SUBAPPLICATION StartStopDemo (* Start/Stop pattern demo: E_SR (persistent start/stop state) gates E_PERMIT, which in turn gates TrueUntil.TRIGGER *)
  (* Standard: 61499-2; Description: Copyright (c) 2026 Meisterschulen am Ostbahnhof This program and the accompanying materials are made available under the terms of the Eclipse Public License 2.0 which is available at https://www.eclipse.org/legal/epl-2.0/ SPDX-License-Identifier: EPL-2.0 *)
  (* Version 1.0, 2026-08-31, Franz Höpfinger, Meisterschulen am Ostbahnhof, Start/Stop design pattern (IEC 61499 primer course, Module 6, Valeriy Vyatkin, slide 70), demo application *)
  PACKAGE Meins::DesingPatterns::StartStopPattern;
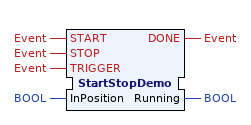
  EVENT_INPUT
    START; (* Start the plant: opens the permit gate *)
    STOP; (* Stop the plant: closes the permit gate *)
    TRIGGER; (* Ask the step to run - only actually reaches it while the plant is started *)
  END_EVENT
  EVENT_OUTPUT
    DONE; (* The step completed (only fires if the plant was started when TRIGGER arrived) *)
  END_EVENT
  VAR_INPUT
    InPosition : BOOL; (* Demo: simulate the step's actuator reaching its position *)
  END_VAR
  VAR_OUTPUT
    Running : BOOL; (* Current start/stop state (E_SR.Q): TRUE while the plant is started *)
  END_VAR
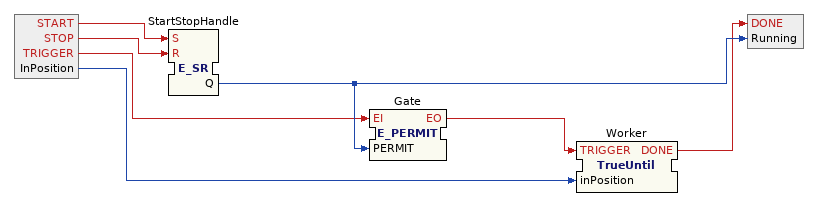
  FBS
    StartStopHandle : iec61499::events::E_SR;
    Gate : iec61499::events::E_PERMIT;
    Worker : Meins::DesingPatterns::ChainOfActionsPattern::TrueUntil;
  END_FBS
  EVENT_CONNECTIONS
    START TO StartStopHandle.S;
    STOP TO StartStopHandle.R;
    TRIGGER TO Gate.EI;
    Gate.EO TO Worker.TRIGGER;
    Worker.DONE TO DONE;
  END_CONNECTIONS
  DATA_CONNECTIONS
    StartStopHandle.Q TO Gate.PERMIT;
    StartStopHandle.Q TO Running;
    InPosition TO Worker.inPosition;
  END_CONNECTIONS
END_SUBAPPLICATION
